(* CODESYS project Simulation_V2.project

Project tree, tasks and I/O mapping:
  Device : CODESYS Virtual Control for Linux SL, CODESYS, order no. 2302000005, version 4.22.0.0
    application Application
      libraries: Standard, 3.5.22.0 (System); VisuDialogs, * (System); Unit Conversion Interfaces, * (Intern); CAA Mathematics, * (CAA Technical Workgroup); SM3_Math, * (CODESYS); SysProcess, * (System); CmpBitmapPool, * (System)
      task MainTask (cyclic, interval t#20ms, priority 1) calls MAIN_PRG, Ablaufkette
      task SoftMotion_PlanningTask (cyclic, interval t#2ms, priority 15) calls nothing
      global variables GVL_OPCUA
      visualisation Topics_Vis
      Structs/
        ST_RobotStatus/
          data type ST_RobotStatus
          data type ST_Pose_Axis
          data type ST_Pose_TCP
        ST_RobotAction/
          data type ST_RobotAction
          data type Error_Codes_RobotAction
        ST_RobotCommand/
          data type ST_RobotCommand
          data type ST_Servo_Axis
          data type ST_Servo_TCP
        ST_Orientierung/
          data type ST_euler
          data type ST_quaternions
      old_code/
        data type Manuell_Achse
        data type TCP_Pose
        program PRG_VISU [ST]
        data type JointState
        FB_Robot/
          function block FB_Robot [FBD]
          function block FB_Watchdog [ST]
          function block FB_RobotCommander [ST]
        Interfaces/
          interface IF_RobotStatus: Ist_Pose_Axis, Ist_Pose_TCP, Ist_Mode, Client_Connection_Status, Update_Watchdog
          interface IF_RobotCommand: Soll_Pose_Axis, Soll_Pose_TCP
        function block FB_Roboter [FBD]: Update_Watchdog, Soll_Pose_Axis, Soll_Pose_TCP, Client_Connection_Status, Ist_Mode, Ist_Pose_Axis, Ist_Pose_TCP
        function block Status_POU [ST]
      program MAIN_PRG [FBD]
      FB_Generell/
        function block FB_MoveAction [ST]: MoveToHome, Ex1_ompl_tcp, Ex2_ompl_joint, Ex3_pilz_tcp_ptp, Ex_4_pilz_tcp_lin, Ablauf_HomePos, Ablauf_Pos1, Ablauf_Pos2, Ablauf_Pos3, Ablauf_Pos4
        function block FB_Modes [FBD]
        function block FB_RobotStatus [ST]
        function block FB_RobotCommand [ST]
      program Ablaufkette [SFC]
      Funktionen/
        function FUNC_quat_to_euler [ST]
        function block FB_Quat_to_ZYZ [FBD]
        function block FB_ZYZ_to_Quat [FBD]
      Symbols
      image pool ImagePool
      global variables GVL_Allg
  libraries: SM3_Robotics, * (CODESYS); VisuSymbols, 4.5.0.0 (System)
  text list GlobalTextList
*)

// Device/Application/old_code/Manuell_Achse
TYPE Manuell_Achse :
STRUCT
	axis_0_plus : BOOL;
	axis_0_minus : BOOL;
	axis_1_plus : BOOL;
	axis_1_minus : BOOL;
	axis_2_plus : BOOL;
	axis_2_minus : BOOL;
	axis_3_plus : BOOL;
	axis_3_minus : BOOL;
	axis_4_plus : BOOL;
	axis_4_minus : BOOL;
	axis_5_plus : BOOL;
	axis_5_minus : BOOL;
	//velocity_spee  einstellen
	//start manuell
END_STRUCT
END_TYPE

// Device/Application/old_code/TCP_Pose
TYPE TCP_Pose :
STRUCT
	trans_x : LREAL;
	trans_y : LREAL;
	trans_z : LREAL;
	rot_x : LREAL;
	rot_y : LREAL;
	rot_z : LREAL;
	rot_w : LREAL;
END_STRUCT
END_TYPE

//TCP Pose in kartesischen Koordinaten
//Rotation wird in quaternions uebermittelt, muss noch umgerechnet werden

// Device/Application/old_code/JointState
TYPE JointState :
STRUCT
	name :ARRAY[0..5] OF STRING;
	position :ARRAY[0..5] OF LREAL; 
	effort :ARRAY[0..5] OF LREAL;
	velocity :ARRAY[0..5] OF LREAL;
END_STRUCT
END_TYPE

// Device/Application/Structs/ST_RobotStatus/ST_RobotStatus
// Gibt den aktuellen Status des Roboters an
TYPE ST_RobotStatus :
STRUCT
	//Joints
	Pos_Axis : ST_Pose_Axis; 	
	
	// TCP mit Orientierung in Quaternions
	Pos_TCP : ST_Pose_TCP;	
	
	//Watchdog
	client_connected : BOOL;
	watchdog_counter : INT;		// Überprüft serverseitige client verbindung
END_STRUCT
END_TYPE

// Device/Application/Structs/ST_RobotCommand/ST_RobotCommand
TYPE ST_RobotCommand :
STRUCT
	// axis manuell
	axis_servo : ST_Servo_Axis;
	
	//tcp manuell
	tcp_servo : ST_Servo_TCP;
	
	//enable: zum starten und stopen der servo_node
	enable : BOOL;
	
	//Watchdog
	client_connected: BOOL;
	watchdog_counter: INT;
END_STRUCT
END_TYPE

// Device/Application/Structs/ST_RobotAction/ST_RobotAction
TYPE ST_RobotAction :
STRUCT
	//Allgemein
	Execute : BOOL;					//Starten der Ausführung (Senden des Goals)
	Error_Code: DINT;				//Feedback ob Ausführung erfolgreich? (Error_code=1)

	//Planer Einstellen
	Motion_Type: STRING;			//string pipeline_id: ompl, pilz_ptp, pilz_lin, pilt_crc
	Planner_ID:STRING;				//string planner_id
	Joint_Goal: BOOL;			
	TCP_GOAL: BOOL;
	num_planning_attempts : DINT;	//int32 num_planning_attempts
	allowed_planning_time: LREAL;	//float64 allowed_planning_time
	max_velocity_scaling: LREAL;		//float64 max_velocity_scaling_factor
	max_acceleration_scaling: LREAL;	//float64 max_acceleration_scaling_factor
	position_tolerance: LREAL;		//float 64 absolute_x_axis_tolerance ->für alle achsen die gleiche toleranz
	orientation_tolerance: LREAL;	//float64
	joint_tolerance : LREAL;
	
	//Joints
	axis_0 : LREAL;		
	axis_1 : LREAL;
	axis_2 : LREAL;
	axis_3 : LREAL;
	axis_4 : LREAL;
	axis_5 : LREAL;
	
	// TCP
	trans_x : LREAL;
	trans_y : LREAL;
	trans_z : LREAL;
	rot_x :  LREAL;
	rot_y : LREAL;
	rot_z : LREAL;
	rot_w : LREAL;
	
	//Watchdog
	client_connected : BOOL;
	watchdog_counter : INT;
END_STRUCT
END_TYPE

// Device/Application/Structs/ST_RobotStatus/ST_Pose_Axis
TYPE ST_Pose_Axis :
STRUCT
	axis_0 : LREAL;
	axis_1 : LREAL;
	axis_2 : LREAL;
	axis_3 : LREAL;
	axis_4 : LREAL;
	axis_5 : LREAL;
END_STRUCT
END_TYPE

// Device/Application/Structs/ST_RobotStatus/ST_Pose_TCP
TYPE ST_Pose_TCP :
STRUCT
	trans_x : LREAL;
	trans_y :  LREAL;
	trans_z : LREAL;
	rot_x : LREAL;
	rot_y : LREAL;
	rot_z : LREAL;
	rot_w : LREAL;
END_STRUCT
END_TYPE

// Device/Application/Structs/ST_RobotCommand/ST_Servo_Axis
TYPE ST_Servo_Axis :
STRUCT
	velocity : LREAL;	
	axis_0 : LREAL;
	axis_1 : LREAL;
	axis_2 : LREAL;
	axis_3 : LREAL;
	axis_4 : LREAL;
	axis_5 : LREAL;
END_STRUCT
END_TYPE

// Device/Application/Structs/ST_RobotCommand/ST_Servo_TCP
TYPE ST_Servo_TCP :
STRUCT
	velocity : LREAL;
	trans_x : LREAL;
	trans_y : LREAL;
	trans_z : LREAL;
	rot_x : LREAL;
	rot_y : LREAL;
	rot_z : LREAL;
	rot_w : LREAL;
END_STRUCT
END_TYPE

// Device/Application/Structs/ST_RobotAction/Error_Codes_RobotAction
{attribute 'qualified_only'}
//{attribute 'strict'}	//CODESYS erlaubt keine TYP Umwandlungen wenn strict aktiv!
{attribute 'to_string'}

TYPE Error_Codes_RobotAction :
(
	NOT_DEFINED := 0,
    SUCCESS := 1,
    FAILURE := 99999,
    PLANNING_FAILED := -1,
    INVALID_MOTION_PLAN := -2,
    MOTION_PLAN_INVALIDATED_BY_ENVIRONMENT_CHANGE := -3,
    CONTROL_FAILED := -4,
    UNABLE_TO_AQUIRE_SENSOR_DATA := -5,
    TIMED_OUT := -6,
    PREEMPTED := -7,
    START_STATE_IN_COLLISION := -10,
    START_STATE_VIOLATES_PATH_CONSTRAINTS := -11,
    START_STATE_INVALID := -26,
    GOAL_IN_COLLISION := -12,
    GOAL_VIOLATES_PATH_CONSTRAINTS := -13,
    GOAL_CONSTRAINTS_VIOLATED := -14,
    GOAL_STATE_INVALID := -27,
    UNRECOGNIZED_GOAL_TYPE := -28,
    INVALID_GROUP_NAME := -15,
    INVALID_GOAL_CONSTRAINTS := -16,
    INVALID_ROBOT_STATE := -17,
    INVALID_LINK_NAME := -18,
    INVALID_OBJECT_NAME := -19,
    FRAME_TRANSFORM_FAILURE := -21,
    COLLISION_CHECKING_UNAVAILABLE := -22,
    ROBOT_STATE_STALE := -23,
    SENSOR_INFO_STALE := -24,
    COMMUNICATION_FAILURE := -25,
    CRASH := -29,
    ABORT := -30,
    NO_IK_SOLUTION := -31
) DINT := NOT_DEFINED;	//Standardwert
END_TYPE

// Device/Application/Structs/ST_Orientierung/ST_euler
//echte Eulerwinkel intrinsich
//ZYZ intrinsisch: bezug auf mitbewegendes Koordinatensystem
//ZYZ extrinsisch: bezug auf festes Koordinatensystem
TYPE ST_euler :
STRUCT
	A : LREAL;	//Z
	B : LREAL;	//Y
	C : LREAL;	//Z
END_STRUCT
END_TYPE

// Device/Application/Structs/ST_Orientierung/ST_quaternions
TYPE ST_quaternions :
STRUCT
	qx: LREAL;
	qy: LREAL;
	qz: LREAL;
	qw: LREAL;
END_STRUCT
END_TYPE

// Device/Application/GVL_OPCUA
{attribute 'qualified_only'}
VAR_GLOBAL
	//Simulation Arm
	//TEST
	//Structs global deklarieren!
	RobotAction: ST_RobotAction;
	RobotStatus : ST_RobotStatus;
	RobotCommand : ST_RobotCommand;
	Execute : BOOL := FALSE;
	
	// Ablaufkette
	TIPP : BOOL; 				// Zum Weiterschalten
	Start_Ablaufkette: BOOL;	// Startet Ablaufkette
	Reset_Ablaufkette: BOOL;	//setzt Schrittkette zurück
	
	//Moveaction 
	Ablauf_HomePos: BOOL;
	Ablauf_Pos1: BOOL;
	Ablauf_Pos2: BOOL;
	Ablauf_Pos3: BOOL;
	Ablauf_Pos4: BOOL;
	
	//Start und Stop per "SoftKeys"
	//Übernimmt ros2 launch ... im docker container
	Start_RViz2 : BOOL;			//Start RViz2
	Stop_RViz2: BOOL;			//Stop RViz2
	Start_OPCClients: BOOL;		//Start OPC Clients
	Stop_OPC_Clients: BOOL;		//Stop OPC Clients
	
END_VAR

VAR_GLOBAL CONSTANT
	PI : REAL := 3.14159;
END_VAR

// Device/Application/GVL_Allg
{attribute 'qualified_only'}
VAR_GLOBAL
	//Action
	rot_A : LREAL;
	rot_B: LREAL;
	rot_C: LREAL;
	
	//mode
END_VAR

// Device/Application/MAIN_PRG
PROGRAM MAIN_PRG
VAR
///////////////////////////////////////////////////		
	//Modus:
	trig: R_TRIG;

	//Objekt RobotAction
	RobotAction: FB_MoveAction;
	// Actions "initialisieren"
	xMoveHome : BOOL;
	xEx1_ompl_tcp: BOOL;
	xEx2_ompl_joint: BOOL;
	xEx3_pilz_tcp_ptp: BOOL;
	xEx4_pilz_tcp_lin: BOOL;
	
	// ENUM für Error Codes
	Status_Error_Codes_Action : Error_Codes_RobotAction;
///////////////////////////////////////////////////	
	
	//Modes
	Modes: FB_Modes;
	
///////////////////////////////////////////////////		

	// ObjektRobotStatus
	RobotStatus: FB_RobotStatus;
	
///////////////////////////////////////////////////	

	//ObjektRobotCommand
	RobotCommand: FB_RobotCommand;
	VIS_Command_axis_0 : LREAL;
	VIS_Command_axis_1 : LREAL;
	VIS_Command_axis_2 : LREAL;
	VIS_Command_axis_3 : LREAL;
	VIS_Command_axis_4 : LREAL;
	VIS_Command_axis_5 : LREAL;
	VIS_Command_axis_velocity : LREAL;
	
	euler : ST_Euler;
	Status_Quat_to_ZYZ: FB_Quat_to_ZYZ;
	Status_ZYZ_to_Quat : FB_ZYZ_to_Quat;
	Action_zyz_to_quat: FB_ZYZ_to_Quat;
END_VAR

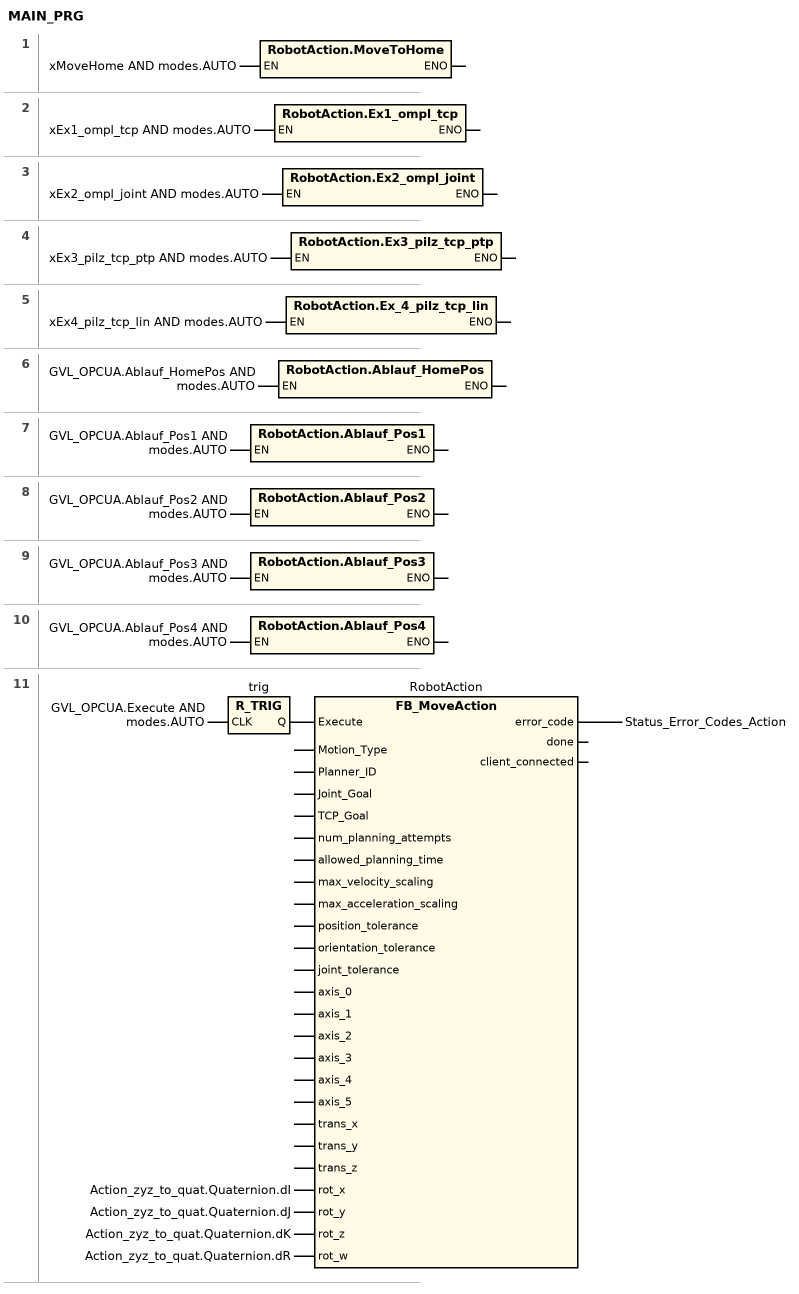
// NETWORK 1
IF xMoveHome AND modes.AUTO THEN RobotAction.MoveToHome(); END_IF

// NETWORK 2
IF xEx1_ompl_tcp AND modes.AUTO THEN RobotAction.Ex1_ompl_tcp(); END_IF

// NETWORK 3
IF xEx2_ompl_joint AND modes.AUTO THEN RobotAction.Ex2_ompl_joint(); END_IF

// NETWORK 4
IF xEx3_pilz_tcp_ptp AND modes.AUTO THEN RobotAction.Ex3_pilz_tcp_ptp(); END_IF

// NETWORK 5
IF xEx4_pilz_tcp_lin AND modes.AUTO THEN RobotAction.Ex_4_pilz_tcp_lin(); END_IF

// NETWORK 6
IF GVL_OPCUA.Ablauf_HomePos AND modes.AUTO THEN RobotAction.Ablauf_HomePos(); END_IF

// NETWORK 7
IF GVL_OPCUA.Ablauf_Pos1 AND modes.AUTO THEN RobotAction.Ablauf_Pos1(); END_IF

// NETWORK 8
IF GVL_OPCUA.Ablauf_Pos2 AND modes.AUTO THEN RobotAction.Ablauf_Pos2(); END_IF

// NETWORK 9
IF GVL_OPCUA.Ablauf_Pos3 AND modes.AUTO THEN RobotAction.Ablauf_Pos3(); END_IF

// NETWORK 10
IF GVL_OPCUA.Ablauf_Pos4 AND modes.AUTO THEN RobotAction.Ablauf_Pos4(); END_IF

// NETWORK 11
trig(CLK := GVL_OPCUA.Execute AND modes.AUTO); // R_TRIG
RobotAction(
    Execute := trig.Q,
    rot_x := Action_zyz_to_quat.Quaternion.dI,
    rot_y := Action_zyz_to_quat.Quaternion.dJ,
    rot_z := Action_zyz_to_quat.Quaternion.dK,
    rot_w := Action_zyz_to_quat.Quaternion.dR); // FB_MoveAction
Status_Error_Codes_Action := RobotAction.error_code;

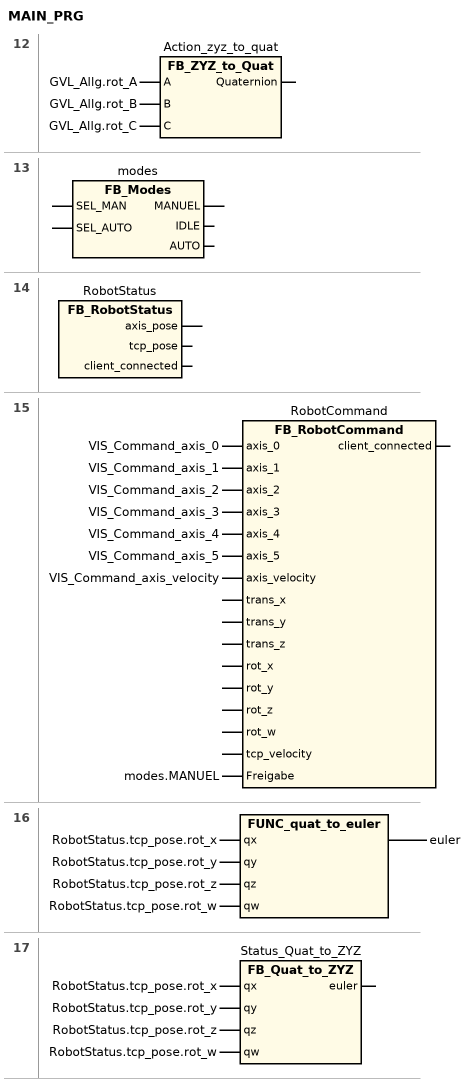
// NETWORK 12
Action_zyz_to_quat(A := GVL_Allg.rot_A, B := GVL_Allg.rot_B, C := GVL_Allg.rot_C); // FB_ZYZ_to_Quat

// NETWORK 13
modes(); // FB_Modes

// NETWORK 14
RobotStatus(); // FB_RobotStatus

// NETWORK 15
RobotCommand(
    axis_0 := VIS_Command_axis_0,
    axis_1 := VIS_Command_axis_1,
    axis_2 := VIS_Command_axis_2,
    axis_3 := VIS_Command_axis_3,
    axis_4 := VIS_Command_axis_4,
    axis_5 := VIS_Command_axis_5,
    axis_velocity := VIS_Command_axis_velocity,
    Freigabe := modes.MANUEL); // FB_RobotCommand

// NETWORK 16
euler := FUNC_quat_to_euler(qx := RobotStatus.tcp_pose.rot_x, qy := RobotStatus.tcp_pose.rot_y, qz := RobotStatus.tcp_pose.rot_z, qw := RobotStatus.tcp_pose.rot_w);

// NETWORK 17
Status_Quat_to_ZYZ(
    qx := RobotStatus.tcp_pose.rot_x,
    qy := RobotStatus.tcp_pose.rot_y,
    qz := RobotStatus.tcp_pose.rot_z,
    qw := RobotStatus.tcp_pose.rot_w); // FB_Quat_to_ZYZ

END_PROGRAM

// Device/Application/FB_Generell/FB_MoveAction
FUNCTION_BLOCK FB_MoveAction
VAR_INPUT
    Execute : BOOL;

    Motion_Type : STRING;
    Planner_ID : STRING;

    Joint_Goal : BOOL;
    TCP_Goal : BOOL;

    num_planning_attempts : DINT;
    allowed_planning_time : LREAL;

    max_velocity_scaling : LREAL;
    max_acceleration_scaling : LREAL;

    position_tolerance : LREAL;
    orientation_tolerance : LREAL;
	joint_tolerance: LREAL;

    // Joints
    axis_0 : LREAL;
    axis_1 : LREAL;
    axis_2 : LREAL;
    axis_3 : LREAL;
    axis_4 : LREAL;
    axis_5 : LREAL;

    // TCP
    trans_x : LREAL;
    trans_y : LREAL;
    trans_z : LREAL;
    rot_x : LREAL;
    rot_y : LREAL;
    rot_z : LREAL;
    rot_w : LREAL;
	
END_VAR
VAR_OUTPUT
	error_code:DINT;
	done : BOOL;
	//Watchdog
	client_connected : BOOL;
END_VAR
VAR
	//Watchdog
	Watchdog_counter : INT;	
	Watchdog_var_old : INT := -1;
	Intervall : TIME :=T#200MS;
	Timer : TON;
	
	//Konvertierung ZYZ->Quat für action
	zyz_to_quat : FB_ZYZ_to_Quat;

END_VAR

// Execute
GVL_OPCUA.RobotAction.Execute := Execute;

// Allgemein
GVL_OPCUA.RobotAction.Motion_Type := Motion_Type;
GVL_OPCUA.RobotAction.Planner_ID := Planner_ID;

GVL_OPCUA.RobotAction.Joint_Goal := Joint_Goal;
GVL_OPCUA.RobotAction.TCP_GOAL := TCP_Goal;

GVL_OPCUA.RobotAction.num_planning_attempts := num_planning_attempts;
GVL_OPCUA.RobotAction.allowed_planning_time := allowed_planning_time;

GVL_OPCUA.RobotAction.max_velocity_scaling := max_velocity_scaling;
GVL_OPCUA.RobotAction.max_acceleration_scaling := max_acceleration_scaling;

GVL_OPCUA.RobotAction.position_tolerance := position_tolerance;
GVL_OPCUA.RobotAction.orientation_tolerance := orientation_tolerance;
GVL_OPCUA.RobotAction.joint_tolerance := joint_tolerance;

// Joints
GVL_OPCUA.RobotAction.axis_0 := axis_0;
GVL_OPCUA.RobotAction.axis_1 := axis_1;
GVL_OPCUA.RobotAction.axis_2 := axis_2;
GVL_OPCUA.RobotAction.axis_3 := axis_3;
GVL_OPCUA.RobotAction.axis_4 := axis_4;
GVL_OPCUA.RobotAction.axis_5 := axis_5;


// TCP
GVL_OPCUA.RobotAction.trans_x := trans_x;
GVL_OPCUA.RobotAction.trans_y := trans_y;
GVL_OPCUA.RobotAction.trans_z := trans_z;

GVL_OPCUA.RobotAction.rot_x := rot_x;
GVL_OPCUA.RobotAction.rot_y := rot_y;
GVL_OPCUA.RobotAction.rot_z := rot_z;
GVL_OPCUA.RobotAction.rot_w := rot_w;

//OUTPUT
error_code := GVL_OPCUA.RobotAction.Error_Code;
IF error_code = 1 THEN
	done := TRUE;
ELSE 
	done := FALSE;
END_IF

//Watchdog
Watchdog_counter := GVL_OPCUA.RobotAction.watchdog_counter;
IF Watchdog_counter <> Watchdog_var_old THEN
	Watchdog_var_old := Watchdog_counter;
	client_connected := TRUE;
	GVL_OPCUA.RobotAction.client_connected := client_connected;
	Timer(IN:=FALSE);

ELSE
	Timer(IN:=TRUE, PT:=Intervall);	
END_IF

IF Timer.Q THEN
	client_connected := FALSE;
	GVL_OPCUA.RobotAction.client_connected := client_connected;
END_IF

ACTION MoveToHome:
//HomePosition
axis_0 := 0.0;
axis_1 := 0.0;
axis_2 := 0.0;
axis_3 := 0.0;
axis_4 := 0.0;
axis_5 := 0.0;
Motion_Type := 'ompl';
Planner_ID := '';
Joint_Goal := TRUE;
TCP_Goal := FALSE;
num_planning_attempts := 10;
allowed_planning_time := 10;
max_velocity_scaling := 0.2;
max_acceleration_scaling := 0.2;
joint_tolerance := 0.01;
END_ACTION

ACTION Ex1_ompl_tcp:
trans_x := 0.114;
trans_y := -0.019;
trans_z := 0.357;
GVL_Allg.rot_A := 0.0;
GVL_Allg.rot_B := 90.0;
GVL_Allg.rot_C := -90.0;
Motion_Type := 'ompl';
Planner_ID := '';
Joint_Goal := FALSE;
TCP_Goal := TRUE;
num_planning_attempts := 10;
allowed_planning_time := 10;
max_velocity_scaling := 0.2;
max_acceleration_scaling := 0.2;
position_tolerance := 0.02;
orientation_tolerance := 0.05;
END_ACTION

ACTION Ex2_ompl_joint:
axis_0 := 0.2;
axis_1 := 0.3;
axis_2 := 0.2;
axis_3 := 0.3;
axis_4 := 0.2;
axis_5 := 0.3;
Motion_Type := 'ompl';
Planner_ID := '';
Joint_Goal := TRUE;
TCP_Goal := FALSE;
num_planning_attempts := 10;
allowed_planning_time := 10;
max_velocity_scaling := 0.2;
max_acceleration_scaling := 0.2;
joint_tolerance := 0.01;
END_ACTION

ACTION Ex3_pilz_tcp_ptp:
trans_x := 0.174;
trans_y := -0.041;
trans_z := 0.244;
GVL_Allg.rot_A := 0.0;
GVL_Allg.rot_B := 90.0;
GVL_Allg.rot_C := -90.0;
Motion_Type := 'pilz_industrial_motion_planner';
Planner_ID := 'PTP';
Joint_Goal := FALSE;
TCP_Goal := TRUE;
num_planning_attempts := 10;
allowed_planning_time := 10;
max_velocity_scaling := 0.05;
max_acceleration_scaling := 0.05;
position_tolerance := 0.02;
orientation_tolerance := 0.05;
END_ACTION

ACTION Ex_4_pilz_tcp_lin:
trans_x := 0.086;
trans_y := -0.086;
trans_z := 0.326;
GVL_Allg.rot_A := 0.0;
GVL_Allg.rot_B := 90.0;
GVL_Allg.rot_C := -90.0;
Motion_Type := 'pilz_industrial_motion_planner';
Planner_ID := 'LIN';
Joint_Goal := FALSE;
TCP_Goal := TRUE;
num_planning_attempts := 10;
allowed_planning_time := 10;
max_velocity_scaling := 0.005;
max_acceleration_scaling := 0.005;
position_tolerance := 0.02;
orientation_tolerance := 0.05;
END_ACTION

ACTION Ablauf_HomePos:
axis_0 := 0.1076;
axis_1 := -0.0931;
axis_2 := -1.667;
axis_3 := 1.773;
axis_4 := 0.07;
axis_5 := 0.19;
Motion_Type := 'ompl';
Planner_ID := '';
Joint_Goal := TRUE;
TCP_Goal := FALSE;
num_planning_attempts := 10;
allowed_planning_time := 10;
max_velocity_scaling := 0.2;
max_acceleration_scaling := 0.2;
joint_tolerance := 0.01;
END_ACTION

ACTION Ablauf_Pos1:
trans_x := 0.1848;
trans_y := -0.0449;
trans_z := 0.2971;

GVL_Allg.rot_A := 0.0;
GVL_Allg.rot_B := 90.0;
GVL_Allg.rot_C := -90.0;

Motion_Type := 'ompl';
Planner_ID := '';
Joint_Goal := FALSE;
TCP_Goal := TRUE;
num_planning_attempts := 10;
allowed_planning_time := 10;
max_velocity_scaling := 0.1;
max_acceleration_scaling := 0.1;
position_tolerance := 0.005;
orientation_tolerance := 0.05;
END_ACTION

ACTION Ablauf_Pos2:
trans_x := 0.1848;
trans_y := -0.0449;
trans_z := 0.2371;
GVL_Allg.rot_A := 0.0;
GVL_Allg.rot_B := 90.0;
GVL_Allg.rot_C := -90.0;
Motion_Type := 'pilz_industrial_motion_planner';
Planner_ID := 'PTP';
Joint_Goal := FALSE;
TCP_Goal := TRUE;
num_planning_attempts := 10;
allowed_planning_time := 10;
max_velocity_scaling := 0.1;
max_acceleration_scaling := 0.1;
position_tolerance := 0.005;
orientation_tolerance := 0.05;
END_ACTION

ACTION Ablauf_Pos3:
trans_x := 0.1248;
trans_y := -0.0449;
trans_z := 0.237;
GVL_Allg.rot_A := 0.0;
GVL_Allg.rot_B := 90.0;
GVL_Allg.rot_C := -90.0;
Motion_Type := 'pilz_industrial_motion_planner';
Planner_ID := 'PTP';
Joint_Goal := FALSE;
TCP_Goal := TRUE;
num_planning_attempts := 10;
allowed_planning_time := 10;
max_velocity_scaling := 0.1;
max_acceleration_scaling := 0.1;
position_tolerance := 0.005;
orientation_tolerance := 0.05;
END_ACTION

ACTION Ablauf_Pos4:
trans_x := 0.1248;
trans_y := -0.0449;
trans_z := 0.2971;
GVL_Allg.rot_A := 0.0;
GVL_Allg.rot_B := 90.0;
GVL_Allg.rot_C := -90.0;
//zyz_to_quat.A:=0.0;
//zyz_to_quat.B :=90.0;
//zyz_to_quat.C := 0.0;
//zyz_to_quat();

//rot_x := zyz_to_quat.Quaternion.dI;
//rot_y := zyz_to_quat.Quaternion.dJ;
//rot_z := zyz_to_quat.Quaternion.dK;
//rot_w := zyz_to_quat.Quaternion.dR;
Motion_Type := 'ompl';
Planner_ID := '';
Joint_Goal := FALSE;
TCP_Goal := TRUE;
num_planning_attempts := 10;
allowed_planning_time := 10;
max_velocity_scaling := 0.1;
max_acceleration_scaling := 0.1;
position_tolerance := 0.005;
orientation_tolerance := 0.05;
END_ACTION

END_FUNCTION_BLOCK

// Device/Application/Funktionen/FB_ZYZ_to_Quat
FUNCTION_BLOCK FB_ZYZ_to_Quat
VAR_INPUT
	A : LREAL;
	B: LREAL;
	C: LREAL;
END_VAR
VAR_OUTPUT
	Quaternion: SMC_Quat;
END_VAR
VAR
	Rotation_Matrix: SMC_Matrix3;
END_VAR

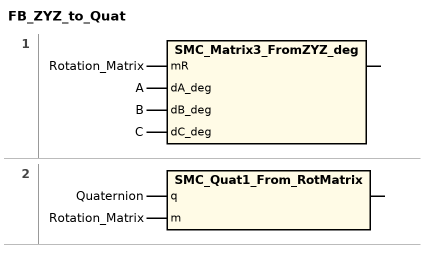
// NETWORK 1
SMC_Matrix3_FromZYZ_deg(mR := Rotation_Matrix, dA_deg := A, dB_deg := B, dC_deg := C);

// NETWORK 2
SMC_Quat1_From_RotMatrix(q := Quaternion, m := Rotation_Matrix);

END_FUNCTION_BLOCK

// Device/Application/FB_Generell/FB_Modes
FUNCTION_BLOCK FB_Modes	//mit Betriebsartenhierachie MAN > AUTO
VAR_INPUT
	SEL_MAN : BOOL;
	SEL_AUTO: BOOL;
END_VAR
VAR_OUTPUT
	MANUEL : BOOL;	//z1
	IDLE: BOOL;		//z0
	AUTO: BOOL;		//z2
END_VAR
VAR
	z0, z1, z2 : BOOL;
	H1, H2: RS;
	z: INT;
END_VAR
VAR // added by the converter: edge detectors and wires of the graphical bodies
    _w1, _w2, _w3 : BOOL;
END_VAR

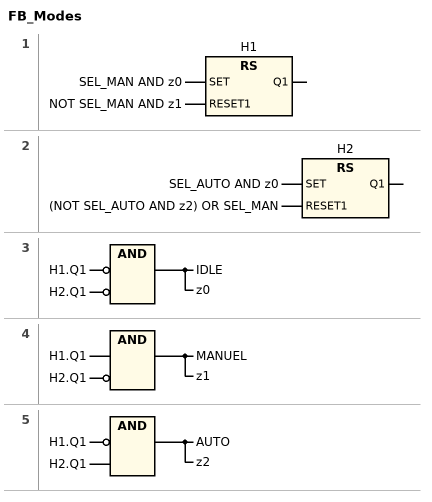
// NETWORK 1
H1(SET := SEL_MAN AND z0, RESET1 := NOT SEL_MAN AND z1); // RS

// NETWORK 2
H2(SET := SEL_AUTO AND z0, RESET1 := (NOT SEL_AUTO AND z2) OR SEL_MAN); // RS

// NETWORK 3
_w1 := NOT H1.Q1 AND NOT H2.Q1;
IDLE := _w1;
z0 := _w1;

// NETWORK 4
_w2 := H1.Q1 AND NOT H2.Q1;
MANUEL := _w2;
z1 := _w2;

// NETWORK 5
_w3 := NOT H1.Q1 AND H2.Q1;
AUTO := _w3;
z2 := _w3;

END_FUNCTION_BLOCK

// Device/Application/FB_Generell/FB_RobotStatus
FUNCTION_BLOCK FB_RobotStatus
VAR_INPUT
END_VAR
VAR_OUTPUT
	// Axis pose in rad
	axis_pose : ST_Pose_Axis;
	
	//TCP Posemit Orientierung in Quaternions
	tcp_pose : ST_Pose_TCP;
	
	
	// Watchdog
	client_connected : BOOL;
END_VAR
VAR
	//Watchdog
	Watchdog_counter : INT;	
	Watchdog_var_old : INT := -1;
	Intervall : TIME :=T#200MS;
	Timer : TON;
END_VAR

// Mappping der Variablen der GVL_OPCUA
axis_pose.axis_0 := GVL_OPCUA.RobotStatus.Pos_Axis.axis_0;
axis_pose.axis_1 := GVL_OPCUA.RobotStatus.Pos_Axis.axis_1;
axis_pose.axis_2 := GVL_OPCUA.RobotStatus.Pos_Axis.axis_2;
axis_pose.axis_3 := GVL_OPCUA.RobotStatus.Pos_Axis.axis_3;
axis_pose.axis_4 := GVL_OPCUA.RobotStatus.Pos_Axis.axis_4;
axis_pose.axis_5 := GVL_OPCUA.RobotStatus.Pos_Axis.axis_5;

tcp_pose.trans_x := GVL_OPCUA.RobotStatus.Pos_TCP.trans_x;
tcp_pose.trans_y := GVL_OPCUA.RobotStatus.Pos_TCP.trans_y;
tcp_pose.trans_z := GVL_OPCUA.RobotStatus.Pos_TCP.trans_z;
tcp_pose.rot_x := GVL_OPCUA.RobotStatus.Pos_TCP.rot_x;
tcp_pose.rot_y := GVL_OPCUA.RobotStatus.Pos_TCP.rot_y;
tcp_pose.rot_z := GVL_OPCUA.RobotStatus.Pos_TCP.rot_z;
tcp_pose.rot_w := GVL_OPCUA.RobotStatus.Pos_TCP.rot_w;

//Watchdog zum Testen ob noch mit StatusClient verbunden!
Watchdog_counter := GVL_OPCUA.RobotStatus.watchdog_counter;
IF Watchdog_counter <> Watchdog_var_old THEN
	Watchdog_var_old :=  Watchdog_counter;
    client_connected := TRUE;
	GVL_OPCUA.RobotStatus.client_connected := client_connected;
    Timer(IN := FALSE);

ELSE
    Timer(IN := TRUE,PT := Intervall );
END_IF;

IF Timer.Q THEN
    client_connected := FALSE;
	GVL_OPCUA.RobotStatus.client_connected := client_connected;
END_IF;

END_FUNCTION_BLOCK

// Device/Application/FB_Generell/FB_RobotCommand
FUNCTION_BLOCK FB_RobotCommand
VAR_INPUT
	axis_0 : LREAL;
	axis_1 : LREAL;
	axis_2: LREAL;
	axis_3 : LREAL;
	axis_4 : LREAL;
	axis_5 : LREAL;
	axis_velocity : LREAL;
	
	trans_x : LREAL;
	trans_y : LREAL;
	trans_z : LREAL;
	rot_x : LREAL;
	rot_y : LREAL;
	rot_z : LREAL;
	rot_w : LREAL;
	tcp_velocity : LREAL;
	
	//Allgemein
	Freigabe:BOOL:=FALSE;
	
END_VAR
VAR_OUTPUT
	// Watchdog
	client_connected : BOOL;
END_VAR
VAR
	//Watchdog
	Watchdog_counter : INT;	
	Watchdog_var_old : INT := -1;
	Intervall : TIME :=T#200MS;
	Timer : TON;
END_VAR

IF Freigabe THEN
	GVL_OPCUA.RobotCommand.axis_servo.axis_0 := axis_0;
	GVL_OPCUA.RobotCommand.axis_servo.axis_1 := axis_1;
	GVL_OPCUA.RobotCommand.axis_servo.axis_2 := axis_2;
	GVL_OPCUA.RobotCommand.axis_servo.axis_3 := axis_3;
	GVL_OPCUA.RobotCommand.axis_servo.axis_4 := axis_4;
	GVL_OPCUA.RobotCommand.axis_servo.axis_5 := axis_5;
	GVL_OPCUA.RobotCommand.axis_servo.velocity := axis_velocity;
	
	GVL_OPCUA.RobotCommand.tcp_servo.trans_x := trans_x;
	GVL_OPCUA.RobotCommand.tcp_servo.trans_y := trans_y;
	GVL_OPCUA.RobotCommand.tcp_servo.trans_z := trans_z;
	GVL_OPCUA.RobotCommand.tcp_servo.rot_x := rot_x;
	GVL_OPCUA.RobotCommand.tcp_servo.rot_y := rot_y;
	GVL_OPCUA.RobotCommand.tcp_servo.rot_z := rot_z;
	GVL_OPCUA.RobotCommand.tcp_servo.rot_w := rot_w;
	GVL_OPCUA.RobotCommand.tcp_servo.velocity := tcp_velocity;
	
	// start der /servo_node/start_servo
	GVL_OPCUA.RobotCommand.enable := TRUE;
	
ELSE
	GVL_OPCUA.RobotCommand.enable := FALSE;
END_IF

//Watchdog zum Testen ob noch mit StatusClient verbunden!
Watchdog_counter := GVL_OPCUA.RobotStatus.watchdog_counter;
IF Watchdog_counter <> Watchdog_var_old THEN
	Watchdog_var_old :=  Watchdog_counter;
    client_connected := TRUE;
	GVL_OPCUA.RobotStatus.client_connected := client_connected;
    Timer(IN := FALSE);

ELSE
    Timer(IN := TRUE,PT := Intervall );
END_IF;

IF Timer.Q THEN
    client_connected := FALSE;
	GVL_OPCUA.RobotStatus.client_connected := client_connected;
END_IF;

END_FUNCTION_BLOCK

// Device/Application/Funktionen/FUNC_quat_to_euler
FUNCTION FUNC_quat_to_euler : ST_euler
VAR_INPUT
	qx : LREAL;
	qy : LREAL;
	qz : LREAL;
	qw : LREAL;
END_VAR
VAR
	r11, r12, r13, r21, r22, r23, r31, r32, r33 : LREAL;
	const_epsilon : LREAL := 1.0E-6; // Toleranz für Gimbal Lock
	result : ST_euler;
	
END_VAR

//Quaternion -> Euler mit ZYZ (intrinsisch) 
//Ausgabe der Euler Winkel in Grad
//Rotationsmatrix Quaternion
r11 := 1.0 - 2.0 * (qy*qy + qz*qz);
r12 := 2.0 * (qx*qy - qz*qw);
r13 := 2.0 * (qx*qz + qy*qw);

r21 := 2.0 * (qx*qy + qz*qw);
r22 := 1.0 - 2.0 * (qx*qx + qz*qz);
r23 := 2.0 * (qy*qz - qx*qw);

r31 := 2.0 * (qx*qz - qy*qw);
r32 := 2.0 * (qy*qz + qx*qw);
r33 := 1.0 - 2.0 * (qx*qx + qy*qy);

result.B := MATH.atan2_func(SQRT(r31*r31+r32*r32),r33);

IF result.B < const_epsilon THEN
	//Gimbal Lock Nordpol
	result.A := 0.0;
	result.C := MATH.atan2_func(r21,r11);
	
ELSIF result.B > (MATH.PI - const_epsilon) THEN
	//Gimbal Lock Südpol
	result.A := 0.0;
	result.C := MATH.atan2_func(-r21,-r11);
ELSE
	//normal
	result.A := MATH.atan2_func(r23,r13);
	result.C := MATH.atan2_func(r32,-r31);
	
END_IF

result.A := result.A * (180.0/MATH.PI);
result.B := result.B * (180.0/MATH.PI);
result.C := result.C * (180.0/MATH.PI);

FUNC_quat_to_euler := result;

END_FUNCTION

// Device/Application/Funktionen/FB_Quat_to_ZYZ
FUNCTION_BLOCK FB_Quat_to_ZYZ
VAR_INPUT
	qx : LREAL;
	qy: LREAL;
	qz:LREAL;
	qw : LREAL;

END_VAR
VAR_OUTPUT
	euler : ST_euler;
END_VAR
VAR
	Quaternion: SMC_Quat;
	Rotation_Matrix: SMC_Matrix3;
END_VAR

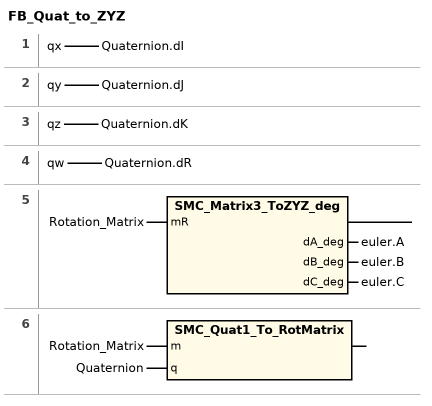
// NETWORK 1
Quaternion.dI := qx;

// NETWORK 2
Quaternion.dJ := qy;

// NETWORK 3
Quaternion.dK := qz;

// NETWORK 4
Quaternion.dR := qw;

// NETWORK 5
SMC_Matrix3_ToZYZ_deg(mR := Rotation_Matrix, dA_deg => euler.A, dB_deg => euler.B, dC_deg => euler.C);

// NETWORK 6
SMC_Quat1_To_RotMatrix(m := Rotation_Matrix, q := Quaternion);

END_FUNCTION_BLOCK

// Device/Application/Ablaufkette
PROGRAM Ablaufkette
VAR
	SFCCurrentStep : STRING;
END_VAR

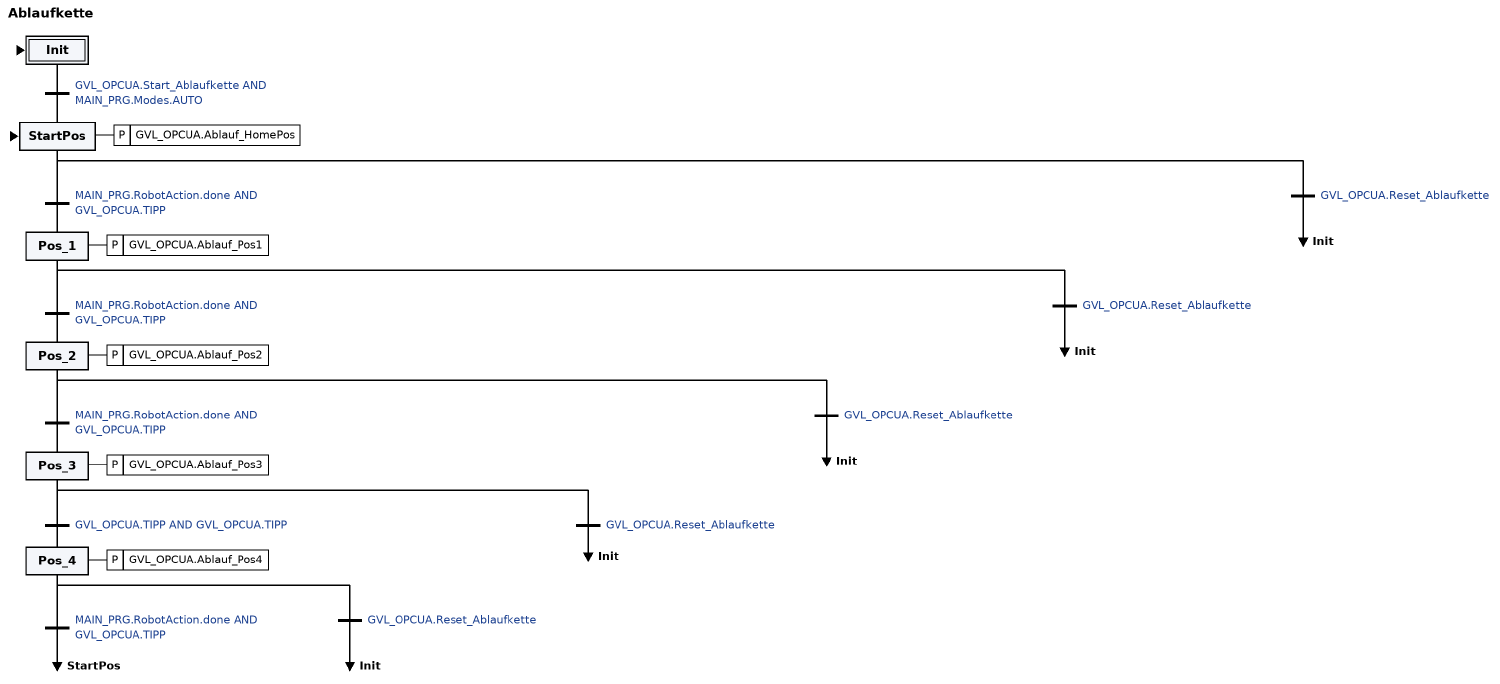
INITIAL_STEP Init:
END_STEP
TRANSITION FROM Init TO StartPos
    := GVL_OPCUA.Start_Ablaufkette AND MAIN_PRG.Modes.AUTO;
END_TRANSITION
STEP StartPos:
    GVL_OPCUA.Ablauf_HomePos(P);
END_STEP
TRANSITION FROM StartPos TO Pos_1
    := MAIN_PRG.RobotAction.done AND GVL_OPCUA.TIPP;
END_TRANSITION
TRANSITION FROM StartPos TO Init
    := GVL_OPCUA.Reset_Ablaufkette;
END_TRANSITION
STEP Pos_1:  // min time t#1s
    GVL_OPCUA.Ablauf_Pos1(P);
END_STEP
TRANSITION FROM Pos_1 TO Pos_2
    := MAIN_PRG.RobotAction.done AND GVL_OPCUA.TIPP;
END_TRANSITION
TRANSITION FROM Pos_1 TO Init
    := GVL_OPCUA.Reset_Ablaufkette;
END_TRANSITION
STEP Pos_2:  // min time t#1s
    GVL_OPCUA.Ablauf_Pos2(P);
END_STEP
TRANSITION FROM Pos_2 TO Pos_3
    := MAIN_PRG.RobotAction.done AND GVL_OPCUA.TIPP;
END_TRANSITION
TRANSITION FROM Pos_2 TO Init
    := GVL_OPCUA.Reset_Ablaufkette;
END_TRANSITION
STEP Pos_3:  // min time t#1s
    GVL_OPCUA.Ablauf_Pos3(P);
END_STEP
TRANSITION FROM Pos_3 TO Pos_4
    := GVL_OPCUA.TIPP AND GVL_OPCUA.TIPP;
END_TRANSITION
TRANSITION FROM Pos_3 TO Init
    := GVL_OPCUA.Reset_Ablaufkette;
END_TRANSITION
STEP Pos_4:  // min time t#1s
    GVL_OPCUA.Ablauf_Pos4(P);
END_STEP
TRANSITION FROM Pos_4 TO StartPos
    := MAIN_PRG.RobotAction.done AND GVL_OPCUA.TIPP;
END_TRANSITION
TRANSITION FROM Pos_4 TO Init
    := GVL_OPCUA.Reset_Ablaufkette;
END_TRANSITION

END_PROGRAM

// Device/Application/old_code/PRG_VISU
PROGRAM PRG_Visu
VAR
    //arrStruct: ARRAY[0..6] OF LREAL;
	Robot : FB_Robot;
	
	//Instanziierung für Roboter
	axis_0_plus :BOOL := FALSE;
	axis_0_minus :BOOL := FALSE;
	axis_1_plus :BOOL := FALSE;
	axis_1_minus :BOOL := FALSE;
	axis_2_plus :BOOL := FALSE;
	axis_2_minus :BOOL := FALSE;
	axis_3_plus :BOOL := FALSE;
	axis_3_minus :BOOL := FALSE;
	axis_4_plus :BOOL := FALSE;
	axis_4_minus :BOOL := FALSE;
	axis_5_plus :BOOL := FALSE;
	axis_5_minus :BOOL := FALSE;
	vis_velocity :LREAL := 0;
END_VAR

Robot();

END_PROGRAM

// Device/Application/old_code/FB_Robot/FB_Robot
FUNCTION_BLOCK FB_Robot
VAR_INPUT
	Command: RobotCommand;
END_VAR
VAR_OUTPUT
	Status: ST_RobotStatus;
END_VAR
VAR
	robotcommand : FB_RobotCommand;
	Watchdog: FB_Watchdog;
END_VAR

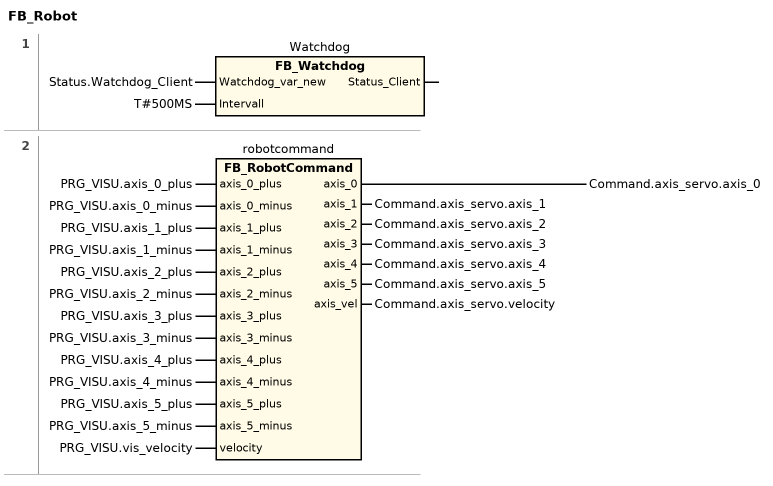
// NETWORK 1
Watchdog(Watchdog_var_new := Status.Watchdog_Client, Intervall := T#500MS); // FB_Watchdog

// NETWORK 2
robotcommand(
    axis_0_plus := PRG_VISU.axis_0_plus,
    axis_0_minus := PRG_VISU.axis_0_minus,
    axis_1_plus := PRG_VISU.axis_1_plus,
    axis_1_minus := PRG_VISU.axis_1_minus,
    axis_2_plus := PRG_VISU.axis_2_plus,
    axis_2_minus := PRG_VISU.axis_2_minus,
    axis_3_plus := PRG_VISU.axis_3_plus,
    axis_3_minus := PRG_VISU.axis_3_minus,
    axis_4_plus := PRG_VISU.axis_4_plus,
    axis_4_minus := PRG_VISU.axis_4_minus,
    axis_5_plus := PRG_VISU.axis_5_plus,
    axis_5_minus := PRG_VISU.axis_5_minus,
    velocity := PRG_VISU.vis_velocity,
    axis_1 => Command.axis_servo.axis_1,
    axis_2 => Command.axis_servo.axis_2,
    axis_3 => Command.axis_servo.axis_3,
    axis_4 => Command.axis_servo.axis_4,
    axis_5 => Command.axis_servo.axis_5,
    axis_vel => Command.axis_servo.velocity); // FB_RobotCommand
Command.axis_servo.axis_0 := robotcommand.axis_0;

END_FUNCTION_BLOCK

// Device/Application/old_code/FB_Robot/FB_Watchdog
FUNCTION_BLOCK FB_Watchdog
VAR_INPUT
	Watchdog_var_new: INT;
	Intervall : TIME;
END_VAR
VAR_OUTPUT
	Status_Client : BOOL;
END_VAR
VAR
	Watchdog_var_old : INT := -1;
	Timer : TON;
END_VAR

IF Watchdog_var_new <> Watchdog_var_old THEN

    Watchdog_var_old := Watchdog_var_new;
    Status_Client := TRUE;
    Timer(IN := FALSE);

ELSE
    Timer(IN := TRUE,PT := Intervall );
END_IF;

IF Timer.Q THEN
    Status_Client := FALSE;
END_IF;

END_FUNCTION_BLOCK

// Device/Application/old_code/FB_Robot/FB_RobotCommander
FUNCTION_BLOCK FB_RobotCommander
VAR_INPUT
	axis_0_plus : BOOL;
	axis_0_minus : BOOL;
	axis_1_plus : BOOL;
	axis_1_minus : BOOL;
	axis_2_plus : BOOL;
	axis_2_minus : BOOL;
	axis_3_plus : BOOL;
	axis_3_minus : BOOL;
	axis_4_plus : BOOL;
	axis_4_minus : BOOL;
	axis_5_plus : BOOL;
	axis_5_minus : BOOL;
	velocity : LREAL;
END_VAR
VAR_OUTPUT
	axis_0 : LREAL;
	axis_1 : LREAL;
	axis_2 : LREAL;
	axis_3 : LREAL;
	axis_4 : LREAL;
	axis_5 : LREAL;
	axis_vel : LREAL;
END_VAR
VAR
END_VAR

// Achse 0
IF axis_0_plus THEN
    axis_0 := 1;
ELSIF axis_0_minus THEN
    axis_0 := -1;
ELSE
    axis_0 := 0;
END_IF;

// Achse 1
IF axis_1_plus THEN
    axis_1 := 1;
ELSIF axis_1_minus THEN
    axis_1 := -1;
ELSE
    axis_1 := 0;
END_IF;

// Achse 2
IF axis_2_plus THEN
    axis_2 := 1;
ELSIF axis_2_minus THEN
    axis_2 := -1;
ELSE
    axis_2 := 0;
END_IF;

// Achse 3
IF axis_3_plus THEN
    axis_3 := 1;
ELSIF axis_3_minus THEN
    axis_3 := -1;
ELSE
    axis_3 := 0;
END_IF;

// Achse 4
IF axis_4_plus THEN
    axis_4 := 1;
ELSIF axis_4_minus THEN
    axis_4 := -1;
ELSE
    axis_4 := 0;
END_IF;

// Achse 5
IF axis_5_plus THEN
    axis_5 := 1;
ELSIF axis_5_minus THEN
    axis_5 := -1;
ELSE
    axis_5 := 0;
END_IF;

// Geschwimdigkeit setzten
axis_vel := velocity;

END_FUNCTION_BLOCK

// Device/Application/old_code/Interfaces/IF_RobotStatus
INTERFACE IF_RobotStatus

PROPERTY Ist_Pose_Axis : ST_Pose_Axis
GET
END_GET
END_PROPERTY

PROPERTY Ist_Pose_TCP : ST_Pose_TCP
GET
END_GET
END_PROPERTY

PROPERTY Ist_Mode : ST_Modes
SET
END_SET
GET
END_GET
END_PROPERTY

PROPERTY Client_Connection_Status : BOOL
SET
END_SET
GET
END_GET
END_PROPERTY

METHOD Update_Watchdog : BOOL
VAR_INPUT
END_VAR
END_METHOD

END_INTERFACE

// Device/Application/old_code/Interfaces/IF_RobotCommand
INTERFACE IF_RobotCommand

PROPERTY Soll_Pose_Axis : ST_Servo_Axis
SET
END_SET
GET
END_GET
END_PROPERTY

PROPERTY Soll_Pose_TCP : ST_Servo_TCP
SET
END_SET
GET
END_GET
END_PROPERTY

END_INTERFACE

// Device/Application/old_code/FB_Roboter
FUNCTION_BLOCK FB_Roboter IMPLEMENTS IF_RobotCommand, IF_RobotStatus
VAR_INPUT
END_VAR
VAR_OUTPUT
END_VAR
VAR
	// --- Command Variablen ---
    _soll_pose_axis : ST_Servo_Axis; // (Passend zu deinem Struct-Namen)
    _soll_pose_tcp  : ST_Servo_TCP;
    
    // --- Status Variablen ---
    _client_connected : BOOL;
    _ist_mode         : ST_Modes;
    _ist_pose_axis    : ST_Pose_Axis;
    _ist_pose_tcp     : ST_Pose_TCP;
END_VAR

// NETWORK 1

{warning 'Methodenimplementierung hinzufügen'}
METHOD Update_Watchdog : BOOL
END_METHOD

{warning 'Eigenschaftenimplementierung hinzufügen'}
PROPERTY Soll_Pose_Axis : ST_Servo_Axis
GET
END_GET
SET
END_SET
END_PROPERTY

{warning 'Eigenschaftenimplementierung hinzufügen'}
PROPERTY Soll_Pose_TCP : ST_Servo_TCP
GET
END_GET
SET
END_SET
END_PROPERTY

{warning 'Eigenschaftenimplementierung hinzufügen'}
PROPERTY Client_Connection_Status : BOOL
GET
END_GET
SET
END_SET
END_PROPERTY

{warning 'Eigenschaftenimplementierung hinzufügen'}
PROPERTY Ist_Mode : ST_Modes
GET
END_GET
SET
END_SET
END_PROPERTY

{warning 'Eigenschaftenimplementierung hinzufügen'}
PROPERTY Ist_Pose_Axis : ST_Pose_Axis
GET
END_GET
SET
END_SET
END_PROPERTY

{warning 'Eigenschaftenimplementierung hinzufügen'}
PROPERTY Ist_Pose_TCP : ST_Pose_TCP
GET
END_GET
SET
END_SET
END_PROPERTY

END_FUNCTION_BLOCK

// Device/Application/old_code/Status_POU
FUNCTION_BLOCK Status_POU
VAR_IN_OUT
END_VAR
VAR_OUTPUT
	Status : ST_RobotStatus;
END_VAR
VAR
END_VAR

END_FUNCTION_BLOCK

// Device/Application/Topics_Vis
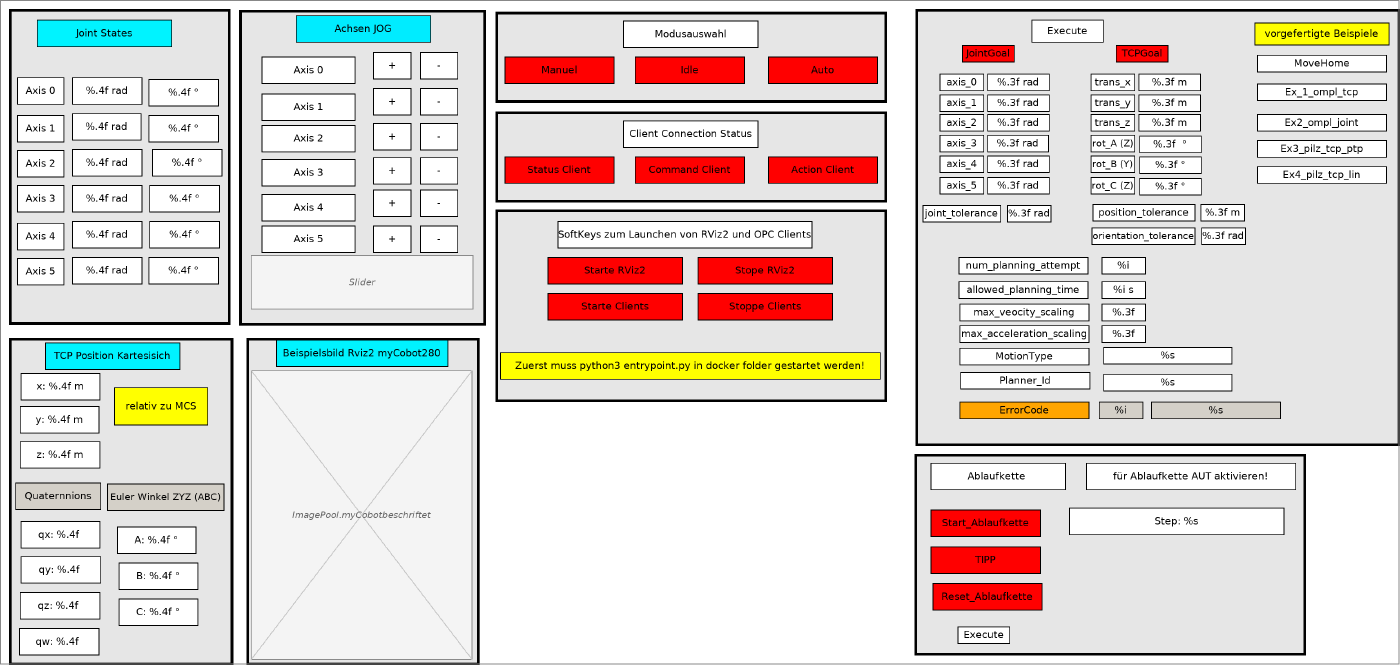
VISUALIZATION Topics_Vis  // 1557x740
    Rectangle (266,11 274x351)
    Rectangle (274,376 259x364)
    Rectangle (551,233 435x214)
    Rectangle (10,376 249x364)
    Rectangle (1018,10 539x486)
    Rectangle (551,13 435x101)
    Rectangle (10,10 246x351)
    Rectangle (41,22 150x30), "Joint States"
    Rectangle (50,381 150x30), "TCP Position Kartesisich"
    Rectangle (23,415 88x30), "x: %.4f m", text variable: MAIN_PRG.RobotStatus.tcp_pose.trans_x
    Rectangle (22,452 88x30), "y: %.4f m", text variable: MAIN_PRG.RobotStatus.tcp_pose.trans_y
    Rectangle (22,491 89x30), "z: %.4f m", text variable: MAIN_PRG.RobotStatus.tcp_pose.trans_z
    Rectangle (23,580 88x30), "qx: %.4f", text variable: MAIN_PRG.RobotStatus.tcp_pose.rot_x
    Rectangle (23,619 89x30), "qy: %.4f", text variable: MAIN_PRG.RobotStatus.tcp_pose.rot_y
    Rectangle (22,659 89x30), "qz: %.4f", text variable: MAIN_PRG.RobotStatus.tcp_pose.rot_z
    Rectangle (21,699 89x30), "qw: %.4f", text variable: MAIN_PRG.RobotStatus.tcp_pose.rot_w
    Rectangle (415,58 42x30), "+"
        OnMouseDown: execute { MAIN_PRG.VIS_Command_axis_0 := +1; }
        OnMouseUp: execute { MAIN_PRG.VIS_Command_axis_0 := 0; }
    Rectangle (467,58 42x30), "-"
        OnMouseDown: execute { MAIN_PRG.VIS_Command_axis_0 := -1; }
        OnMouseUp: execute { MAIN_PRG.VIS_Command_axis_0 := 0; }
    Rectangle (415,98 42x30), "+"
        OnMouseDown: execute { MAIN_PRG.VIS_Command_axis_1 := +1; }
        OnMouseUp: execute { MAIN_PRG.VIS_Command_axis_1 := 0; }
    Rectangle (467,137 42x30), "-"
        OnMouseDown: execute { MAIN_PRG.VIS_Command_axis_2 := -1; }
        OnMouseUp: execute { MAIN_PRG.VIS_Command_axis_2 := 0; }
    Rectangle (415,137 42x30), "+"
        OnMouseDown: execute { MAIN_PRG.VIS_Command_axis_2 := +1; }
        OnMouseUp: execute { MAIN_PRG.VIS_Command_axis_2 := 0; }
    Rectangle (415,175 42x30), "+"
        OnMouseDown: execute { MAIN_PRG.VIS_Command_axis_3 := +1; }
        OnMouseUp: execute { MAIN_PRG.VIS_Command_axis_3 := 0; }
    Rectangle (467,98 42x30), "-"
        OnMouseDown: execute { MAIN_PRG.VIS_Command_axis_1 := -1; }
        OnMouseUp: execute { MAIN_PRG.VIS_Command_axis_1 := 0; }
    Rectangle (467,175 42x30), "-"
        OnMouseDown: execute { MAIN_PRG.VIS_Command_axis_3 := -1; }
        OnMouseUp: execute { MAIN_PRG.VIS_Command_axis_3 := 0; }
    Rectangle (415,211 42x30), "+"
        OnMouseDown: execute { MAIN_PRG.VIS_Command_axis_4 := +1; }
        OnMouseUp: execute { MAIN_PRG.VIS_Command_axis_4 := 0; }
    Rectangle (467,211 42x30), "-"
        OnMouseDown: execute { MAIN_PRG.VIS_Command_axis_4 := -1; }
        OnMouseUp: execute { MAIN_PRG.VIS_Command_axis_4 := 0; }
    Rectangle (415,251 42x30), "+"
        OnMouseDown: execute { MAIN_PRG.VIS_Command_axis_5 := +1; }
        OnMouseUp: execute { MAIN_PRG.VIS_Command_axis_5 := 0; }
    Rectangle (467,251 42x30), "-"
        OnMouseDown: execute { MAIN_PRG.VIS_Command_axis_5 := -1; }
        OnMouseUp: execute { MAIN_PRG.VIS_Command_axis_5 := 0; }
    Slider (279,284 247x60), variable: MAIN_PRG.VIS_Command_axis_velocity, scale 0..1
    Rectangle (693,23 150x30), "Modusauswahl"
    Rectangle (80,86 78x30), "%.4f rad", text variable: MAIN_PRG.RobotStatus.axis_pose.axis_0
    Rectangle (80,126 77x30), "%.4f rad", text variable: MAIN_PRG.RobotStatus.axis_pose.axis_1
    Rectangle (80,166 78x30), "%.4f rad", text variable: MAIN_PRG.RobotStatus.axis_pose.axis_2
    Rectangle (80,206 78x30), "%.4f rad", text variable: MAIN_PRG.RobotStatus.axis_pose.axis_3
    Rectangle (80,246 78x30), "%.4f rad", text variable: MAIN_PRG.RobotStatus.axis_pose.axis_4
    Rectangle (80,286 78x30), "%.4f rad", text variable: MAIN_PRG.RobotStatus.axis_pose.axis_5
    Rectangle (329,17 150x30), "Achsen JOG"
    Rectangle (561,63 122x30), "Manuel", colour toggle: MAIN_PRG.Modes.MANUEL
        toggle MAIN_PRG.Modes.SEL_MAN p2164770859=TRUE
    Rectangle (854,63 122x30), "Auto", colour toggle: MAIN_PRG.Modes.AUTO
        toggle MAIN_PRG.Modes.SEL_AUTO p2164770859=TRUE
    Rectangle (706,63 122x30), "Idle", colour toggle: MAIN_PRG.Modes.IDLE
    Rectangle (1045,82 49x19), "axis_0"
    Rectangle (1045,105 49x19), "axis_1"
    Rectangle (1045,127 49x19), "axis_2"
    Rectangle (1045,150 49x19), "axis_3"
    Rectangle (1045,173 49x19), "axis_4"
    Rectangle (1045,197 49x19), "axis_5"
    Rectangle (1098,82 69x19), "%.3f rad", text variable: MAIN_PRG.RobotAction.axis_0
        OnMouseClick: write the text variable via Default
    Rectangle (1098,105 69x19), "%.3f rad", text variable: MAIN_PRG.RobotAction.axis_1
        OnMouseClick: write the text variable via Default
    Rectangle (1098,127 69x19), "%.3f rad", text variable: MAIN_PRG.RobotAction.axis_2
        OnMouseClick: write the text variable via Default
    Rectangle (1098,150 68x19), "%.3f rad", text variable: MAIN_PRG.RobotAction.axis_3
        OnMouseClick: write the text variable via Default
    Rectangle (1098,173 69x19), "%.3f rad", text variable: MAIN_PRG.RobotAction.axis_4
        OnMouseClick: write the text variable via Default
    Rectangle (1098,197 69x19), "%.3f rad", text variable: MAIN_PRG.RobotAction.axis_5
        OnMouseClick: write the text variable via Default
    Rectangle (1213,82 49x19), "trans_x"
    Rectangle (1213,105 49x19), "trans_y"
    Rectangle (1213,127 49x19), "trans_z"
    Rectangle (1266,82 69x19), "%.3f m", text variable: MAIN_PRG.RobotAction.trans_x
        OnMouseClick: write the text variable via Default
    Rectangle (1266,105 69x19), "%.3f m", text variable: MAIN_PRG.RobotAction.trans_y
        OnMouseClick: write the text variable via Default
    Rectangle (1266,127 69x19), "%.3f m", text variable: MAIN_PRG.RobotAction.trans_z
        OnMouseClick: write the text variable via Default
    Rectangle (1147,22 80x25), "Execute"
        tap GVL_OPCUA.Execute
    Rectangle (1070,50 58x19), "JointGoal", colour toggle: MAIN_PRG.RobotAction.Joint_Goal
        toggle MAIN_PRG.RobotAction.Joint_Goal
    Rectangle (1241,50 58x19), "TCPGoal", colour toggle: MAIN_PRG.RobotAction.TCP_Goal
        toggle MAIN_PRG.RobotAction.TCP_Goal
    Rectangle (1066,286 144x19), "num_planning_attempt"
    Rectangle (1066,313 144x19), "allowed_planning_time"
    Rectangle (1067,338 144x19), "max_veocity_scaling"
    Rectangle (1067,362 144x19), "max_acceleration_scaling"
    Rectangle (1215,227 114x19), "position_tolerance"
    Rectangle (1214,253 115x19), "orientation_tolerance"
    Rectangle (1225,286 49x19), "%i", text variable: MAIN_PRG.RobotAction.num_planning_attempts
        OnMouseClick: write the text variable via Default
    Rectangle (1225,313 49x19), "%i s", text variable: MAIN_PRG.RobotAction.allowed_planning_time
        OnMouseClick: write the text variable via Default
    Rectangle (1225,338 49x19), "%.3f", text variable: MAIN_PRG.RobotAction.max_velocity_scaling
        OnMouseClick: write the text variable via Default
    Rectangle (1225,362 49x19), "%.3f", text variable: MAIN_PRG.RobotAction.max_acceleration_scaling
        OnMouseClick: write the text variable via Default
    Rectangle (1335,227 49x19), "%.3f m", text variable: MAIN_PRG.RobotAction.position_tolerance
        OnMouseClick: write the text variable via Default
    Rectangle (1336,253 49x19), "%.3f rad", text variable: MAIN_PRG.RobotAction.orientation_tolerance
        OnMouseClick: write the text variable via Default
    Rectangle (1067,387 144x19), "MotionType"
    Rectangle (1068,414 144x19), "Planner_Id"
    Rectangle (1067,447 144x19), "ErrorCode"
    Rectangle (1222,447 49x19), "%i", text variable: MAIN_PRG.RobotAction.error_code
    Rectangle (1227,386 143x19), "%s", text variable: MAIN_PRG.RobotAction.Motion_Type
        OnMouseClick: write the text variable via Default
    Rectangle (1227,416 143x19), "%s", text variable: MAIN_PRG.RobotAction.Planner_ID
        OnMouseClick: write the text variable via Default
    Rectangle (1398,61 144x19), "MoveHome"
        tap MAIN_PRG.xMoveHome
    Rectangle (1280,447 144x19), "%s", text variable: MAIN_PRG.Status_Error_Codes_Action
    Rectangle (551,124 435x101)
    Rectangle (693,134 150x30), "Client Connection Status"
    Rectangle (561,174 122x30), "Status Client", colour toggle: MAIN_PRG.RobotStatus.client_connected
    Rectangle (854,174 122x30), "Action Client", colour toggle: MAIN_PRG.RobotAction.client_connected
    Rectangle (706,174 122x30), "Command Client", colour toggle: MAIN_PRG.RobotCommand.client_connected
    Rectangle (1398,93 144x19), "Ex_1_ompl_tcp"
        tap MAIN_PRG.xEx1_ompl_tcp
    Rectangle (1398,127 144x19), "Ex2_ompl_joint"
        tap MAIN_PRG.xEx2_ompl_joint
    Rectangle (1398,156 144x19), "Ex3_pilz_tcp_ptp"
        tap MAIN_PRG.xEx3_pilz_tcp_ptp
    Rectangle (1398,185 144x19), "Ex4_pilz_tcp_lin"
        tap MAIN_PRG.xEx4_pilz_tcp_lin
    Rectangle (165,88 78x30), "%.4f °", text variable: MAIN_PRG.RobotStatus.axis_pose.axis_0 *(180.0/GVL_OPCUA.PI)
    Rectangle (165,128 78x30), "%.4f °", text variable: MAIN_PRG.RobotStatus.axis_pose.axis_1 *(180.0/GVL_OPCUA.PI)
    Rectangle (169,166 78x30), "%.4f °", text variable: MAIN_PRG.RobotStatus.axis_pose.axis_2 *(180.0/GVL_OPCUA.PI)
    Rectangle (166,206 78x30), "%.4f °", text variable: MAIN_PRG.RobotStatus.axis_pose.axis_3 *(180.0/GVL_OPCUA.PI)
    Rectangle (166,246 78x30), "%.4f °", text variable: MAIN_PRG.RobotStatus.axis_pose.axis_4 *(180.0/GVL_OPCUA.PI)
    Rectangle (165,286 78x30), "%.4f °", text variable: MAIN_PRG.RobotStatus.axis_pose.axis_5 *(180.0/GVL_OPCUA.PI)
    Rectangle (130,586 88x30), "A: %.4f °", text variable: MAIN_PRG.euler.A
    Rectangle (132,626 88x30), "B: %.4f °", text variable: MAIN_PRG.euler.B
    Rectangle (132,666 88x30), "C: %.4f °", text variable: MAIN_PRG.euler.C
    Rectangle (119,538 130x30), "Euler Winkel ZYZ (ABC)"
    Rectangle (1017,505 435x224)
    Rectangle (1035,515 150x30), "Ablaufkette"
    Rectangle (1035,608 122x30), "TIPP", colour toggle: MAIN_PRG.RobotStatus.client_connected
        tap GVL_OPCUA.TIPP
    Rectangle (1035,567 122x30), "Start_Ablaufkette", colour toggle: MAIN_PRG.RobotStatus.client_connected
        tap GVL_OPCUA.Start_Ablaufkette
    Rectangle (1189,565 239x30), "Step: %s", text variable: Ablaufkette.SFCCurrentStep
    Rectangle (1208,515 233x30), "für Ablaufkette AUT aktivieren!"
    Rectangle (1037,649 122x30), "Reset_Ablaufkette", colour toggle: MAIN_PRG.RobotStatus.client_connected
        tap GVL_OPCUA.Reset_Ablaufkette
    Rectangle (1065,697 58x19), "Execute"
        tap GVL_OPCUA.Execute
    Rectangle (17,537 95x30), "Quaternnions"
    Rectangle (609,286 150x30), "Starte RViz2"
        toggle GVL_OPCUA.Start_RViz2
    Rectangle (609,326 150x30), "Starte Clients"
        toggle GVL_OPCUA.Start_OPCClients
    Rectangle (776,326 150x30), "Stoppe Clients"
        toggle GVL_OPCUA.Stop_OPC_Clients
    Rectangle (776,286 150x30), "Stope RViz2"
        toggle GVL_OPCUA.Stop_RViz2
    Rectangle (291,63 104x30), "Axis 0"
    Rectangle (291,104 104x30), "Axis 1"
    Rectangle (291,139 104x30), "Axis 2"
    Rectangle (291,177 104x30), "Axis 3"
    Rectangle (291,216 104x30), "Axis 4"
    Rectangle (291,251 104x30), "Axis 5"
    Rectangle (19,86 52x30), "Axis 0"
    Rectangle (19,128 52x30), "Axis 1"
    Rectangle (19,167 52x30), "Axis 2"
    Rectangle (19,206 52x30), "Axis 3"
    Rectangle (19,248 52x30), "Axis 4"
    Rectangle (19,287 52x30), "Axis 5"
    RoundedRectangle (127,431 104x42), "relativ zu MCS"
    Image (279,412 246x322), image: ImagePool.myCobotbeschriftet
    Rectangle (307,378 191x30), "Beispielsbild Rviz2 myCobot280"
    RoundedRectangle (1395,25 150x25), "vorgefertigte Beispiele"
    Rectangle (620,246 283x30), "SoftKeys zum Launchen von RViz2 und OPC Clients"
    Rectangle (556,392 423x30), "Zuerst muss python3 entrypoint.py in docker folder gestartet werden!"
    Rectangle (1213,150 49x19), "rot_A (Z)"
    Rectangle (1213,173 49x19), "rot_B (Y)"
    Rectangle (1213,197 49x19), "rot_C (Z)"
    Rectangle (1267,151 69x19), "%.3f °", text variable: GVL_Allg.rot_A
        OnMouseClick: write the text variable via Default
    Rectangle (1267,174 69x19), "%.3f °", text variable: GVL_Allg.rot_B
        OnMouseClick: write the text variable via Default
    Rectangle (1267,198 69x19), "%.3f °", text variable: GVL_Allg.rot_C
        OnMouseClick: write the text variable via Default
    Rectangle (1026,228 87x19), "joint_tolerance"
    Rectangle (1120,228 49x19), "%.3f rad", text variable: MAIN_PRG.RobotAction.joint_tolerance
        OnMouseClick: write the text variable via Default
END_VISUALIZATION
